// TIA Portal project "array_ile_indirect_adresleme" (V18)

(* hardware
DEVICE "S7-1200 station_1"  S7-1200 Station
   slot 0: "Rack_0"  S7-1200 Rack  Rack  V1.0
   slot 1: "PLC_1"  CPU 1214C DC/DC/DC  6ES7 214-1AG40-0XB0  V4.6
*)

// ===== PLC "PLC_1"  CPU 1214C DC/DC/DC =====

VAR_GLOBAL   // PLC tag table "Default tag table"
   "Tag_1" AT %I0.0 : Bool;
   "Tag_2" AT %M22.2 : Bool;
   "Tag_3" AT %IW64 : Word;
   "Tag_4" AT %MD10 : DInt;
END_VAR

DATA_BLOCK "KAZAN"   // DB1
{ S7_Optimized_Access := 'TRUE' }
VERSION : 0.1
   VAR
      SICAKLIK : Array[0..15] of Int;
   END_VAR
BEGIN
END_DATA_BLOCK

// folder: System blocks/Program resources

DATA_BLOCK "SAYICI"   // DB2
{ S7_Optimized_Access := 'TRUE' }
AUTHOR : Simatic
FAMILY : IEC
NAME : CNTR
VERSION : 1.0
// stored: InstanceOfName IEC_COUNTER
"IEC_COUNTER"
BEGIN
END_DATA_BLOCK

// folder: (top level)

FUNCTION "Block_1" : Void   // FC1, LAD
{ S7_Optimized_Access := 'TRUE' }
VERSION : 0.1
   VAR_TEMP
      SAYI : Int;
   END_VAR
BEGIN

REGION Network 1
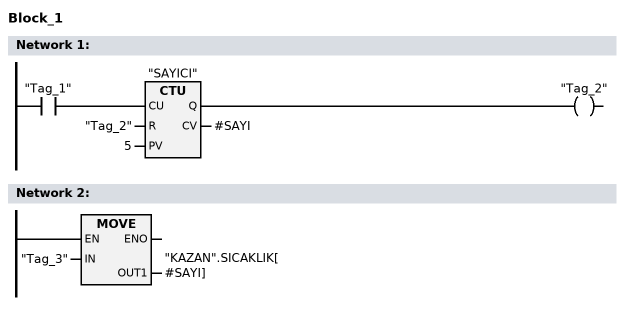
   "SAYICI".CTU(CU := "Tag_1", R := "Tag_2", PV := 5, CV => #SAYI);
   "Tag_2" := "SAYICI".Q;
END_REGION

REGION Network 2
   RUNG wire#powerrail
      Move(in := "Tag_3", out1 => "KAZAN".SICAKLIK[#SAYI])
   END_RUNG
   // the same network as SCL:
   "KAZAN".SICAKLIK[#SAYI] := "Tag_3";
END_REGION
END_FUNCTION

ORGANIZATION_BLOCK "Main"   // OB1, LAD, ProgramCycle
TITLE = "Main Program Sweep (Cycle)"
{ S7_Optimized_Access := 'TRUE' }
VERSION : 0.1
   VAR_INPUT
      Initial_Call : Bool;   // Initial call of this OB
      Remanence : Bool;   // =True, if remanent data are available
   END_VAR
BEGIN

REGION Network 1
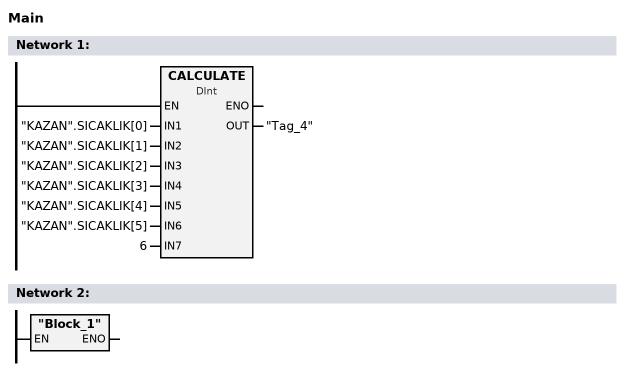
   RUNG wire#powerrail
      { S7_Templates := "SrcType := DInt"; S7_Expression := "(IN1+IN2+IN3+IN4+IN5+IN6)/IN7" } Calculate(in1 := "KAZAN".SICAKLIK[0], in2 := "KAZAN".SICAKLIK[1], in3 := "KAZAN".SICAKLIK[2], in4 := "KAZAN".SICAKLIK[3], in5 := "KAZAN".SICAKLIK[4], in6 := "KAZAN".SICAKLIK[5], in7 := 6, out => "Tag_4")
   END_RUNG
   // the same network as SCL:
   "Tag_4" := ("KAZAN".SICAKLIK[0]+"KAZAN".SICAKLIK[1]+"KAZAN".SICAKLIK[2]+"KAZAN".SICAKLIK[3]+"KAZAN".SICAKLIK[4]+"KAZAN".SICAKLIK[5])/6;
END_REGION

REGION Network 2
   RUNG wire#powerrail
      "Block_1"()
   END_RUNG
   // the same network as SCL:
   "Block_1"();
END_REGION
END_ORGANIZATION_BLOCK